# EPICS autosave request: iocBoot/iocAH501/auto_settings.req
file "quadEM_settings.req",            P=$(P), R=$(R)
file "quadEM_Plugin_settings.req",     P=$(P), R=$(R)
